TYPE st_FlowBaseCore :
STRUCT
  Start:BOOL;
  Excute:BOOL;
  Done:BOOL;
END_STRUCT
END_TYPE

(* stored: Version 1.1.0.1, ProductVersion 3.1.4024.13
   DUT st_FlowBaseCore: Id {8575d881-a0c2-4250-b97c-eaf119f06ec6} *)
